// TIA Portal V17 export
// export: Created 2023-12-22T15:28:36.1567415Z, ExportSetting WithDefaults, DisplayName Totally Integrated Automation Portal, DisplayVersion V17, DisplayName TIA Portal Openness, DisplayVersion V17, DisplayName TIA Portal Version Control Interface, DisplayVersion V17, DisplayName STEP 7 Professional, DisplayVersion V17, DisplayName STEP 7 Safety, DisplayVersion V17, DisplayName WinCC Advanced, DisplayVersion V17
DATA_BLOCK "M_DA_example_DB"   // DB600
VERSION : 0.1
// stored: AutoNumber false, DBAccessibleFromOPCUA true, InstanceOfName DRV_M_DA, InstanceOfType FB
"DRV_M_DA"
   // VAR_INPUT
   //    All_Block : Bool;
   // END_VAR
   // VAR_IN_OUT
   //    FB_QF : Bool;
   //    FB_KM : Bool;
   //    S_Alarm : Bool;
   //    CMD_Run : Bool;
   // END_VAR
   // VAR RETAIN
   //    CMD : "CMD";
   //    Mode : Int;
   //    Status : Int;
   //    Use : Struct
   //       QF { S7_SetPoint := 'True'} : Bool;
   //       KM { S7_SetPoint := 'True'} : Bool;
   //       OpTime { S7_SetPoint := 'True'} : Bool;
   //       Analog { S7_SetPoint := 'True'} : Bool;
   //       Local_Keys : Bool;
   //    END_STRUCT;
   //    FB : Struct
   //       QF : Bool;
   //       KM : Bool;
   //       Local_Start : Bool;
   //       Local_Stop : Bool;
   //    END_STRUCT;
   //    ON : Bool;
   //    OFF : Bool;
   //    Tx { S7_SetPoint := 'True'} : Array[0..3] of "Time_S";
   //    Inv : Struct
   //       CMD { S7_SetPoint := 'True'} : Bool;
   //       QF { S7_SetPoint := 'True'} : Bool;
   //       KM { S7_SetPoint := 'True'} : Bool;
   //    END_STRUCT;
   //    Alarm : Struct
   //       Block : Bool;
   //       QF : Bool;
   //       Start : Bool;
   //       Stop : Bool;
   //       Termo : Bool;
   //       Alarm : Bool;
   //       Safety : Bool;
   //       OpTime : Bool;
   //    END_STRUCT;
   //    Alarms : Word;
   //    Events : Word;
   //    pos : Array[0..15] of Bool;
   //    OpTime_h : DInt;
   //    OpTime_s { S7_SetPoint := 'True'} : DInt;
   //    OpTime_SP { S7_SetPoint := 'True'} : DInt;
   //    OpTime_Now_h : DInt;
   //    OpTime_Now_s { S7_SetPoint := 'True'} : DInt;
   //    CodeID { S7_SetPoint := 'True'} : Int;
   //    Indirect : Struct
   //       FB_QF { S7_SetPoint := 'True'} : Bool;
   //       FB_KM { S7_SetPoint := 'True'} : Bool;
   //       CMD { S7_SetPoint := 'True'} : Bool;
   //    END_STRUCT;
   //    Indirect_BYTE : Struct
   //       FB_QF { S7_SetPoint := 'True'} : Int;
   //       FB_KM { S7_SetPoint := 'True'} : Int;
   //       CMD { S7_SetPoint := 'True'} : Int;
   //    END_STRUCT;
   //    Indirect_BIT : Struct
   //       FB_QF { S7_SetPoint := 'True'} : Int;
   //       FB_KM { S7_SetPoint := 'True'} : Int;
   //       CMD { S7_SetPoint := 'True'} : Int;
   //    END_STRUCT;
   //    SP_A : Real;
   //    SP_M : Real;
   //    ADDR { S7_SetPoint := 'True'} : Int;
   //    Converter { S7_SetPoint := 'True'} : "Converter";
   //    VmA : Real;
   //    Output_Type { S7_SetPoint := 'True'} : Int;
   //    "Type" { S7_SetPoint := 'True'} : Int;
   //    Slow { S7_SetPoint := 'True'} : "Slow";
   //    Time_DTL { S7_SetPoint := 'True'} : DTL;
   // END_VAR
BEGIN
END_DATA_BLOCK
